// SIMATIC S7-200 SMART project (STEP 7-Micro/WIN SMART), CPU ST60

SYMBOL_TABLE 系统符号
First_Scan_On    SM0.1    // 仅在第一个扫描周期时接通
END_SYMBOL_TABLE

ORGANIZATION_BLOCK MAIN:OB1
TITLE=程序注释
BEGIN
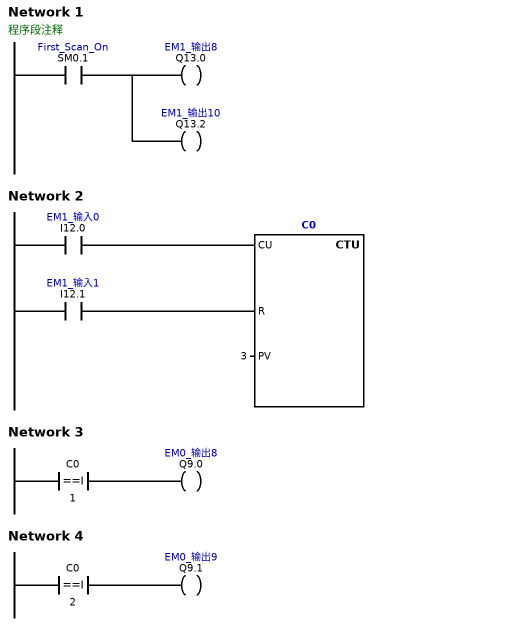
Network 1
// 程序段注释
LD     First_Scan_On:SM0.1
=      EM1_输出8:Q13.0
=      EM1_输出10:Q13.2
Network 2
LD     EM1_输入0:I12.0
LD     EM1_输入1:I12.1
CTU    C0, 3
Network 3
LDW=   C0, 1
=      EM0_输出8:Q9.0
Network 4
LDW=   C0, 2
=      EM0_输出9:Q9.1
END_ORGANIZATION_BLOCK
